TYPE M3Tabs :
(
	OVERVIEW := 0,
    ROTATION := 1,
    TRANSLATION := 2,
    IO := 3,
    CONFIG := 4
);
END_TYPE

(* stored: Version 1.1.0.1, ProductVersion 3.1.4018.2
   DUT M3Tabs: Id {35438742-45e7-4a03-8daf-6ffd37df0047} *)
